// TIA Portal V20 export
DATA_BLOCK "ShiftInitBools"   // DB257
// stored: MemoryReserve 100
   VAR
      earlyShift : Bool;
      lateShift : Bool;
      nightShift : Bool;
   END_VAR
BEGIN
END_DATA_BLOCK
